{attribute 'linkalways'}
{attribute 'no_explicit_call' := 'do not call this POU directly'}
{attribute 'enable_dynamic_creation'}
FUNCTION_BLOCK QueueNode IMPLEMENTS I_QueueNode
VAR
	internalBuffer : POINTER TO BYTE;
	internalBufferSize : UDINT;
	nextNode : I_QueueNode;
END_VAR

METHOD PRIVATE CopyInternalBufferToDestination
VAR_INPUT
	DestinationAddress : PVOID;
END_VAR
memcpy(DestinationAddress,internalBuffer,internalBufferSize);
END_METHOD

METHOD PRIVATE CopySourceToInternalBuffer
VAR_INPUT
	SourceAddress : PVOID;
END_VAR
memcpy(internalBuffer,SourceAddress,internalBufferSize);
END_METHOD

METHOD PRIVATE DeleteInternalBuffer
IF internalBuffer <> 0 THEN
	__DELETE(internalBuffer);
END_IF
END_METHOD

METHOD PUBLIC Destroy
VAR_INPUT
END_VAR
DeleteInternalBuffer();
__Delete(this);
END_METHOD

METHOD FB_init : BOOL
VAR_INPUT
	bInitRetains : BOOL; // if TRUE, the retain variables are initialized (warm start / cold start)
	bInCopyCode : BOOL;  // if TRUE, the instance afterwards gets moved into the copy code (online change)
	Source : ANY;
END_VAR
MakeInternalBufferOfSize(DINT_TO_UDINT(Source.diSize));
CopySourceToInternalBuffer(Source.pValue);
END_METHOD

METHOD PUBLIC Get : BOOL;
VAR_INPUT
	Destination : ANY;
END_VAR
IF NOT IsInternalBufferSameSizeAs(DINT_TO_UDINT(Destination.diSize)) THEN
	RETURN;
END_IF

CopyInternalBufferToDestination(Destination.pValue);
END_METHOD

METHOD PRIVATE IsInternalBufferSameSizeAs : BOOL
VAR_INPUT
	Size : UDINT;
END_VAR
IF internalBuffer = 0 THEN
	RETURN;
END_IF

IF internalBufferSize <> Size THEN
	RETURN;
END_IF

IsInternalBufferSameSizeAs := TRUE;
END_METHOD

METHOD PRIVATE MakeInternalBufferOfSize
VAR_INPUT
	Size : UDINT;
END_VAR
internalBufferSize := Size;
internalBuffer := __NEW(BYTE, internalBufferSize);
END_METHOD

PROPERTY PUBLIC Next : I_QueueNode
GET
Next := nextNode;
END_GET
SET // PUBLIC
nextNode := Next;
END_SET
END_PROPERTY

END_FUNCTION_BLOCK

(* stored: Version 1.1.0.1, ProductVersion 3.1.4024.11
   POU QueueNode: Id {5727fc62-2cdf-415b-88d9-0a182275d5b3}, SpecialFunc None
   Folder Constructor: Id {99d07663-8d19-444c-b251-386e086d188e}
   Folder Private: Id {8bc744f6-366f-4502-91dd-8a6e8367ac86}
   Method CopyInternalBufferToDestination: Id {435865c6-abf1-4aa0-a18b-a0a4ddf72f61}
   Method CopySourceToInternalBuffer: Id {6750840f-f21a-4729-9758-5829588ca080}
   Method DeleteInternalBuffer: Id {9d425e50-5d59-4bce-ac65-98e7adb2fa57}
   Method Destroy: Id {52151c94-c18b-4c21-b66f-3c84449673c0}
   Method FB_init: Id {8f96ec32-be93-451a-9997-77c5ca2fa316}
   Method Get: Id {9d220e81-9b34-496e-ba7e-f8a9c727acaa}
   Method IsInternalBufferSameSizeAs: Id {df860d3d-74b9-4d0c-af51-1d764004b71e}
   Method MakeInternalBufferOfSize: Id {8a46851a-86e2-41f9-8e05-dc45af79cb58}
   Property Next: Id {8e1ddf3a-4b70-487f-b591-2b5bcaf89b07}
   Get Get: Id {46ce132e-8357-4d98-8acf-9c947d626300}
   Set Set: Id {f2ac2e7c-d2be-4808-906e-c82174eb21b6} *)
